FUNCTION_BLOCK FB_PersistentDataManager
VAR_INPUT
END_VAR
VAR_OUTPUT
END_VAR
VAR
	FbWritePersistentData : FB_WritePersistentData ;
	cmdWrite : BOOL := FALSE ;
	TOfWriteInterval	: TOf ;
	CmdWriteFromTime	: BOOL ; 
	TestjeWritten		: BOOL ;
END_VAR

// ===== persistent write interval =====
 TOfWriteInterval(	IN := cmdWrite OR NOT TOfWriteInterval.Q,
	 				PT	:= T#5M  );

IF NOT TOfWriteInterval.Q THEN 
	cmdWrite := TRUE ;
END_IF

// ===== write persistent data =====
	FbWritePersistentData ( PORT 	:= 851,
							START 	:= CmdWrite,
							TMOUT 	:= T#1S,	
							mode 	:= E_PersistentMode.SPDM_VAR_BOOST );	

IF cmdWrite AND FbWritePersistentData.BUSY THEN 
	cmdWrite := FALSE ;
END_IF

METHOD PUBLIC Write : BOOL
VAR_INPUT
END_VAR
IF NOT FbWritePersistentData.BUSY THEN 
	cmdWrite := TRUE ;
ELSE 
	Write := TRUE ;
END_IF
END_METHOD

END_FUNCTION_BLOCK

(* stored: Version 1.1.0.1, ProductVersion 3.1.4024.11
   POU FB_PersistentDataManager: Id {5c72dac1-9833-4672-b715-b19477d15b62}, SpecialFunc None
   Method Write: Id {19a5b35c-c9d0-4c73-b29c-5c39d2c6be4f} *)
